FUNCTION REAL_TO_STRING2 : string
VAR_INPUT
	rIn: LREAL;
	nDigits: BYTE;
END_VAR
VAR
	nMult: DINT := 1;
	nI: BYTE;
END_VAR

FOR nI:=1 TO nDigits DO
	nMult:=nMult*10;
END_FOR
REAL_TO_STRING2:=LREAL_TO_STRING(DINT_TO_LREAL(LREAL_TO_DINT(rIn*nMult))/nMult);

END_FUNCTION

(* stored: Version 1.1.0.1, ProductVersion 3.1.4020.3
   POU REAL_TO_STRING2: Id {6d0f9c79-04f3-4a33-bd87-e8c27c6c01cd}, SpecialFunc None *)
